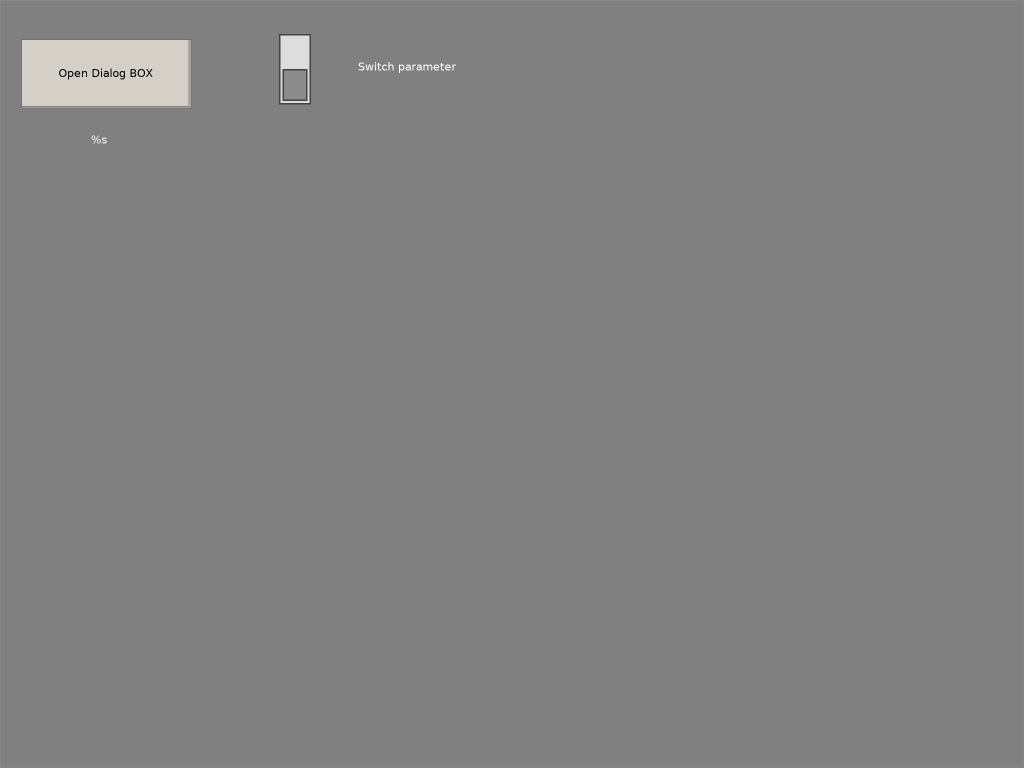
VISUALIZATION Visualization2  // 1024x768
    Button (21,39 170x69), "Open Dialog BOX"
        tap P_Dialog.bOpen
    Rectangle (24,125 150x30), "%s", text variable: P_Dialog.sResult, invisible if: Not P_Dialog.bVisible
    DipSwitch (260,34 70x70), variable: P_Dialog.bSwitchParameter, behaviour: TOGGLE, style: Switch-DipSwitch-Gray
    Label (332,52 150x30), "Switch parameter"
END_VISUALIZATION

(* stored: Version 1.1.0.1, ProductVersion 3.1.4024.3
   Visu Visualization2: Id {81fa2fbb-ac67-4cda-bd49-d7cee9863cab} *)
